FUNCTION_BLOCK FB_QuantityLREALPublic EXTENDS FB_FalliblePublic IMPLEMENTS I_QuantityLREALPublic
VAR
    {attribute 'pytmc' := '
        pv: Value
        io: io
        field: DESC Value of quantity.
    '}
    fValue : LREAL;

    {attribute 'pytmc' := '
        pv: Units
        io: io
        field: DESC Units of quantity.
    '}
    sUnits : T_MaxString;
END_VAR


METHOD Copy
VAR_INPUT
    QuantityToCopy : I_QuantityLREAL;
END_VAR

Val := QuantityToCopy.Val;
Units := QuantityToCopy.Units;

IF QuantityToCopy.GetError() THEN
    SetError(Msg := QuantityToCopy.GetErrorMsg());
ELSE
    ClearError();
END_IF
END_METHOD


METHOD FB_Init: BOOL
VAR_INPUT
    bInitRetains: BOOL; // TRUE: the retain variables are initialized (reset warm / reset cold)
    bInCopyCode: BOOL;  // TRUE: the instance will be copied to the copy code afterward (online change)

    Units : T_MaxString;
END_VAR

THIS^.Units := Units;
END_METHOD


PROPERTY Units : T_MaxString
GET

Units := sUnits;
END_GET
SET

sUnits := Units;
END_SET
END_PROPERTY


PROPERTY Val : LREAL
GET

Val := fValue;
END_GET
SET

fValue := Val;
END_SET
END_PROPERTY

END_FUNCTION_BLOCK

(* stored: Version 1.1.0.1
   POU FB_QuantityLREALPublic: Id {61a079b2-6c1c-4fd2-8539-4d329186c818}, SpecialFunc None
   Method Copy: Id {e9a16c39-fdfb-48f8-b851-f88bccf51c70}
   Method FB_Init: Id {7bc0b41b-56c9-4e5b-8420-077118483cd8}
   Property Units: Id {1cb8fb78-a36e-4512-8f0d-9859fb13e09b}
   Get Get: Id {b7745cbb-f60c-4e2f-a574-b085908c7700}
   Set Set: Id {cce0cfd5-9583-48ea-b1b0-530adb61858b}
   Property Val: Id {c3a58fd7-0f36-4895-8dca-e917000fa2c5}
   Get Get: Id {434e5f80-9d1b-414e-a8ec-5f5fbb7c883b}
   Set Set: Id {d5064fb1-a3bf-467a-a596-8b3f646c000d} *)
